FUNCTION_BLOCK FB_WaitCommand IMPLEMENTS I_Command
VAR
END_VAR

{attribute 'monitoring' := 'call'}
PROPERTY Description : STRING
GET
Description := _Description;
END_GET
END_PROPERTY

METHOD Execute : E_Progress
CASE _Target OF
	
	E_ValvePosition.Home:
		_Valve.MoveToHome();
	
	E_ValvePosition.Work:
		_Valve.MoveToWork();
END_CASE

Execute := E_Progress.Completed;
END_METHOD

//FB_Init is always available implicitly and it is used primarily for initialization.
//The return value is not evaluated. For a specific influence, you can also declare the
//methods explicitly and provide additional code there with the standard initialization
//code. You can evaluate the return value.
METHOD FB_Init: BOOL
VAR_INPUT
    bInitRetains: BOOL; // TRUE: the retain variables are initialized (reset warm / reset cold)
    bInCopyCode: BOOL;  // TRUE: the instance will be copied to the copy code afterward (online change)   
	
	minWaitTime : TIME;
	maxWaitTime : TIME;
	condition : FB_Condition?;
END_VAR
_Valve := valve;
_Target := target;
_Description := description;
END_METHOD

METHOD Reset
VAR_INPUT
END_VAR
// nothing to reset here
END_METHOD

END_FUNCTION_BLOCK

(* stored: Version 1.1.0.1
   POU FB_WaitCommand: Id {ee48ed06-d6a4-4427-864b-5735a143195c}, SpecialFunc None
   Property Description: Id {cf856734-5e67-4fbd-9acd-5eef8430cea2}
   Get Get: Id {9606a3b8-9c11-45da-bee8-7b4b3879e4b2}
   Method Execute: Id {243712fe-f590-4562-ad4c-e6ae33e5faa2}
   Method FB_Init: Id {1d072f35-2629-4a18-ad97-2c5b48ff9410}
   Method Reset: Id {5042e983-7f4a-45b2-b0cd-c26e70af9285} *)
